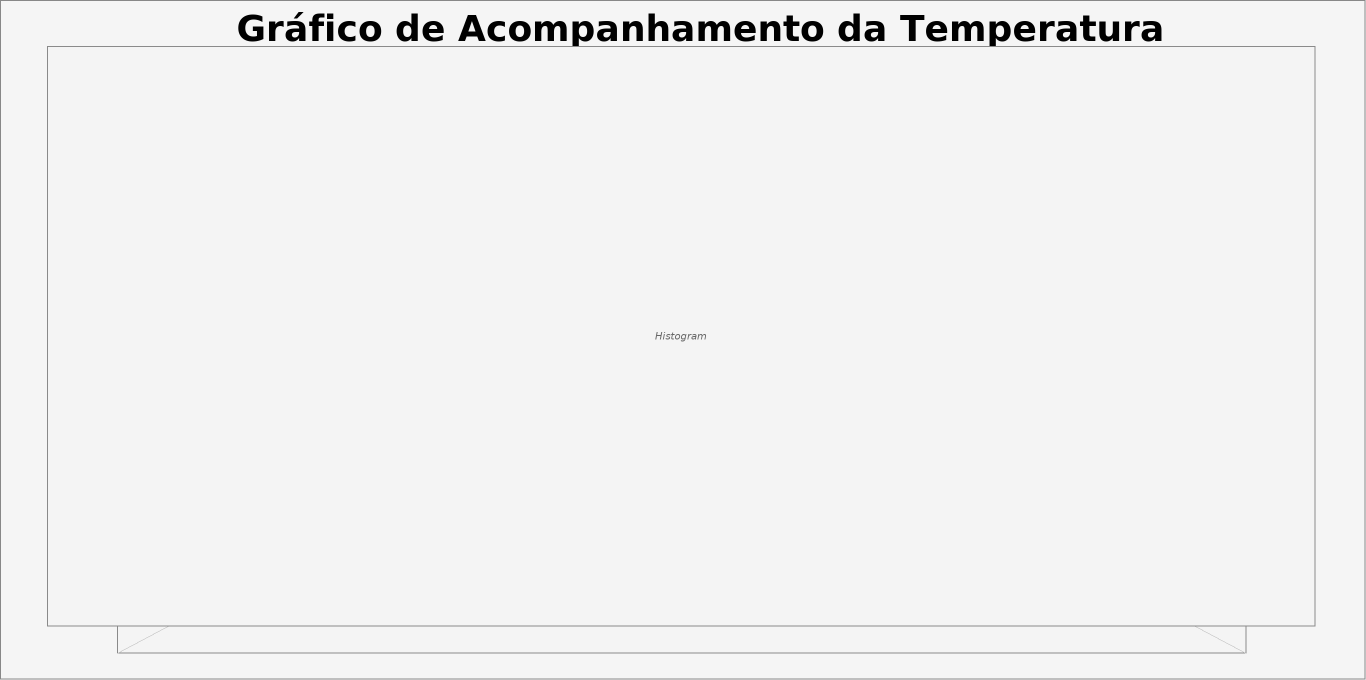
VISUALIZATION Grafico_2  // 1366x680
    Image (117,53 1129x600), image: ImagePool.teseagraf
    Histogram (47,46 1268x580), scale format: %.1f, scale 0..150
        p1518820177: GVL_P.arrTempVisu020
        p102497268: GVL_P.arrTempVisu020
        p788070771: ARRAY [1..720] OF REAL
    Label (262,7 877x43), "Gráfico de Acompanhamento da Temperatura"
    Histogram (47,46 1268x580), scale format: %.1f, scale 0..150
        p1518820177: GVL_P.arrTemp020
        p102497268: GVL_P.arrTemp020
        p788070771: ARRAY [1..720] OF REAL
END_VISUALIZATION

(* stored: Version 1.1.0.1, ProductVersion 3.1.4024.12
   Visu Grafico_2: Id {6fbf8b98-0a47-4fda-bebc-650f6e070dee} *)
